ADAPTER AdapterType (* Adapter Interface *)
  (* Standard: 61499-1 *)
  (* Version 0.2, 2003-12-05, JHC, Rockwell Automation, Changed name from NEWADAPTER *)
  (* Version 0.1, 2002-01-08, JHC, Rockwell Automation, Added IND/RSP, renamed data, added sequences. *)
  (* Version 0.0, 2000-05-27, JHC, Rockwell Automation *)
  (* Compiler header: package fb.rt.template; *)
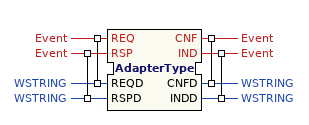
  EVENT_INPUT
    REQ WITH REQD; (* Request from Socket *)
    RSP WITH RSPD; (* Response from Socket *)
  END_EVENT
  EVENT_OUTPUT
    CNF WITH CNFD; (* Confirmation from Plug *)
    IND WITH INDD; (* Indication from Plug *)
  END_EVENT
  VAR_INPUT
    REQD : WSTRING; (* Request Data from Socket *)
    RSPD : WSTRING; (* Response Data from Socket *)
  END_VAR
  VAR_OUTPUT
    CNFD : WSTRING; (* Confirmation Data from Plug *)
    INDD : WSTRING; (* Indication Data from Plug *)
  END_VAR
  SERVICE SOCKET/PLUG
    SEQUENCE request_confirm
      SOCKET.REQ(REQD) -> PLUG.REQ(REQD);
      PLUG.CNF(CNFD) -> SOCKET.CNF(CNFD);
    END_SEQUENCE
    SEQUENCE indication_response
      PLUG.IND(INDD) -> SOCKET.IND(INDD);
      SOCKET.RSP(RSPD) -> PLUG.RSP(RSPD);
    END_SEQUENCE
  END_SERVICE
END_ADAPTER
